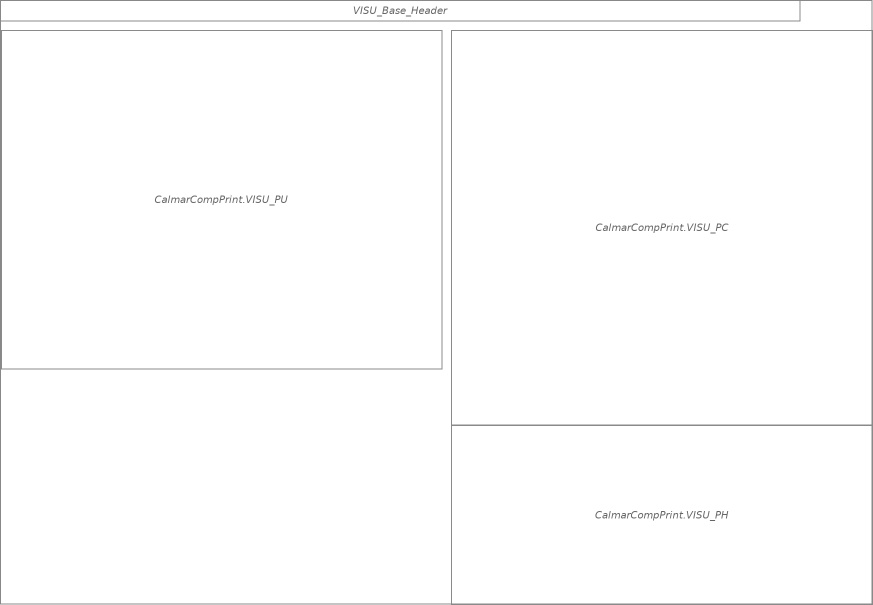
VISUALIZATION VISU_PRINT  // 873x605
    Frame (451,30 422x395)
        shows CalmarCompPrint.VISU_PC(m_visu_fb := PRG_PRINT.fb_visu_pc)
    Frame (1,30 441x339)
        shows CalmarCompPrint.VISU_PU(m_visu_fb := PRG_PRINT.fb_visu_pu)
    Frame (451,425 422x180)
        shows CalmarCompPrint.VISU_PH(m_visu_fb := PRG_PRINT.fb_visu_ph)
    Frame (0,0 800x21)
        shows VISU_Base_Header()
END_VISUALIZATION

(* stored: Version 1.1.0.1, ProductVersion 3.1.4024.9
   Visu VISU_PRINT: Id {5989a128-84ed-4a3d-84aa-3fbdeb85974a} *)
